{attribute 'qualified_only'}
VAR_GLOBAL
	fbJson : FB_JsonSaxWriter;
END_VAR

(* stored: Version 1.1.0.1
   GVL PMPS_TOOLS: Id {72c6e40b-919b-47ae-b308-65c949e33cfe} *)
